INTERFACE ITF_SubsystemTransportEmulation EXTENDS __System.IQueryInterface

METHOD M_CallInterface : BOOL
END_METHOD

METHOD M_GetTransportData : REFERENCE TO ST_TransportDataEmulation
END_METHOD

METHOD M_Init : BOOL
VAR_INPUT
	mInit			: BOOL; // Force init
END_VAR
END_METHOD

METHOD M_MoveTU_DataIndex : DINT
END_METHOD

END_INTERFACE

(* stored: Version 1.1.0.1, ProductVersion 3.1.4022.12
   Itf ITF_SubsystemTransportEmulation: Id {d5895885-a7f5-4f15-8f94-9ff110ddc5b8}
   Method M_CallInterface: Id {01fa0f83-2a17-4744-9eaf-1c941ac0eff7}
   Method M_GetTransportData: Id {fdc1b644-402c-49e4-bc91-11a8ec349d77}
   Method M_Init: Id {db48107b-a0b5-4de7-9b1e-0176033af18a}
   Method M_MoveTU_DataIndex: Id {d3e0bc9b-9a68-4650-a59c-afdda58ea3cd} *)
